{attribute 'qualified_only' := ''}
{attribute 'strict' := ''}
TYPE AXIS_STATUS :
(
	ErrorStop := 0,
	Disabled := 1,
	Stopping := 2,
	Homing := 3,
	Standstill := 4,
	DiscreteMotion := 5,
	ContinuousMotion := 6,
	SynchronizedMotion := 7
);
END_TYPE

(* stored: Version 1.1.0.1, ProductVersion 3.1.4024.11
   DUT AXIS_STATUS: Id {49fa1d5e-a2a4-4ae7-aa5b-b6affe5a3b60} *)
